FUNCTION_BLOCK FB_BagCloser
VAR_INPUT
  ams_net_id: STRING;
END_VAR
VAR_OUTPUT
END_VAR
VAR
	// Variable to be read from the app in python.
	status: BagMachineStatus;
	//bag_detection_status: BagDetectionStatus;
	bag_holder_status: BagHolderStatus;
	bag_status: BagStatus;
	current_bag_cmd: BagCmd;
	current_bag_height_status: BagHeightStatus;

	adsread				: ADSREAD;
	adswrite			: ADSWRITE;
	iMethodTest			: BagMachineStatus;
	bagCloseStatus 		: BagMachineStatus;
  	error_code			: UINT;

	adsArr				: AdsArr;
	iAds				: INT;
	ton_ms				: TON;

	iMachineStatus		: INT;//inArr[0]
	iBagStatus			: INT;//inArr[1]
END_VAR

	adsread(
			NETID:=ams_net_id , 
			PORT:=851 , 
			IDXGRP:=16#00004020 , 
			IDXOFFS:=100 , 
			LEN:= SIZEOF(adsArr.inArr), 
			DESTADDR:= ADR(adsArr.inArr), 
			READ:=, 
			TMOUT:=T#2S , 
			BUSY=> , 
			ERR=> , 
			ERRID=> );
	adswrite(
			NETID:=ams_net_id , 
			PORT:=851, 
			IDXGRP:=16#00004020, 
			IDXOFFS:=200, 
			LEN:=SIZEOF(adsArr.outArr) , 
			SRCADDR:=ADR(adsArr.outArr) , 
			WRITE:= , 
			TMOUT:=T#2S , 
			BUSY=> , 
			ERR=> , 
			ERRID=> );
ton_ms(PT:=T#2MS);			
CASE iAds OF 
	0:
		adsread.READ	:= FALSE;
		adswrite.WRITE	:= FALSE;	
		iAds	:=1;
	1:
		ton_ms.IN	:= TRUE;
		IF ton_ms.Q THEN
			ton_ms.IN	:= FALSE;
			iAds	:=2;
		END_IF
	2:
		adsread.READ	:= TRUE;
		adswrite.WRITE	:= TRUE;
		iAds	:=3;
	3:
		ton_ms.IN	:= TRUE;
		IF ton_ms.Q THEN
			ton_ms.IN	:= FALSE;
			iAds	:=0;
		END_IF	
END_CASE
//inputArr:
//		[0]:machine status;
//		[1]:bag status;
//		[2]:fixture status
//outputArr:
//		[0]:line status;
//		[1]:bag cmd(0: do_nothing, 1:take_bag,2:bag_done_unclamping;);
//		[2]:height detect cmd(0:idle,1:ok,2:ng)
iMachineStatus	:= WORD_TO_INT(adsArr.inArr[0]);
iBagStatus := WORD_TO_INT(adsArr.inArr[1]);
 
adsArr.outArr[1]	:= INT_TO_WORD(current_bag_cmd);
adsArr.outArr[2]	:= INT_TO_WORD(current_bag_height_status);

CASE adsArr.inArr[0] OF
	0:status	:= BagMachineStatus.OFF;
	1:status	:= BagMachineStatus.BUSY;
	2:status	:= BagMachineStatus.READY;
	3:status	:= BagMachineStatus.RESET;
	4:status	:= BagMachineStatus.ERROR;
	5:status	:= BagMachineStatus.STOPPED;
END_CASE
CASE adsArr.inArr[1] OF
	0:bag_status	:= BagStatus.UNKNOWN;
	1:bag_status	:= BagStatus.READY;
	2:bag_status	:= BagStatus.INSERTED;
	3:bag_status	:= BagStatus.REMOVED;
END_CASE
CASE adsArr.inArr[2] OF
	0:bag_holder_status	:= BagHolderStatus.UNKNOWN;
	1:bag_holder_status	:= BagHolderStatus.DOWN;
	2:bag_holder_status	:= BagHolderStatus.UP;
END_CASE

CASE current_bag_cmd OF
	BagCmd.DO_NOTHING:
		;
	BagCmd.INSERT_BAG_HOLDER:
		IF fixture_ready() THEN
			current_bag_cmd	:=0;
		END_IF		
	BagCmd.REMOVE_BAG_HOLDER:
		IF bag_done_unclamping() THEN
			current_bag_cmd	:=0;
		END_IF	
	BagCmd.STOP:
		current_bag_cmd	:= BagCmd.STOP;
		IF status = BagMachineStatus.STOPPED THEN
			current_bag_cmd	:= BagCmd.DO_NOTHING;
		END_IF
		
END_CASE

{attribute 'TcRpcEnable'}
METHOD PUBLIC bag_done_unclamping : BOOL
VAR_INPUT

END_VAR
bag_done_unclamping	:= FALSE;
current_bag_cmd	:= BagCmd.REMOVE_BAG_HOLDER;
IF bag_removed OR unload_ready THEN //avoid not catch signal of removed
	bag_done_unclamping := TRUE;
	current_bag_cmd	:= BagCmd.DO_NOTHING;
END_IF
END_METHOD

PROPERTY bag_removed : BOOL
GET
bag_removed	:= (WORD_TO_INT(adsArr.inArr[1])	= BagStatus.REMOVED);
END_GET
END_PROPERTY

{attribute 'TcRpcEnable'}
METHOD PUBLIC fixture_ready : BOOL
VAR_INPUT

END_VAR
fixture_ready	:= FALSE;
current_bag_cmd	:= BagCmd.INSERT_BAG_HOLDER;
IF machine_inserted THEN
	fixture_ready	:= TRUE;
	current_bag_cmd	:= 	BagCmd.DO_NOTHING;
END_IF
END_METHOD

METHOD M_Init : BOOL
VAR_INPUT
END_VAR
M_Init	:= FALSE;
current_bag_cmd	:= BagCmd.DO_NOTHING;
current_bag_height_status := BagHeightStatus.UNKNOWN;
M_Init	:= TRUE;
END_METHOD

PROPERTY machine_inserted : BOOL
GET
machine_inserted	:= (WORD_TO_INT(adsArr.inArr[1])	= BagStatus.INSERTED);
END_GET
END_PROPERTY

PROPERTY unload_ready : BOOL
GET
unload_ready	:= (WORD_TO_INT(adsArr.inArr[1])	= BagStatus.READY);
END_GET
END_PROPERTY

END_FUNCTION_BLOCK

(* stored: Version 1.1.0.1, ProductVersion 3.1.4024.12
   POU FB_BagCloser: Id {678bc602-a9e5-4e7d-94ba-1a138b16ef52}, SpecialFunc None
   Method bag_done_unclamping: Id {e047a4f5-01c2-4724-98d7-fd4c5489bb8e}
   Property bag_removed: Id {42fdd4c2-b1b0-40fd-b9d0-6bc8b59e8947}
   Get Get: Id {d52869db-1d62-4dd3-96ce-888cb2f81a29}
   Method fixture_ready: Id {38c86974-e5a7-4331-a074-f2b44f4137b9}
   Method M_Init: Id {c7122a50-0b88-4965-9082-2579505fb32a}
   Property machine_inserted: Id {8b3bbd2f-7f3d-4679-9bd2-27237076212b}
   Get Get: Id {70820c96-6148-49c5-a139-06a614438dd7}
   Property unload_ready: Id {c36c0a27-bfee-4b89-9e12-141da2b9c8c6}
   Get Get: Id {b0b68d0c-36a7-4abb-b777-e5a55260dddb} *)
